FUNCTION_BLOCK Fb_FaultHandler
VAR_INPUT
END_VAR
VAR_OUTPUT
	arActiveFaults 	: ARRAY [0..Param_Messages.nMAX_MESSAGES_SHOWN] OF UDT_Fault  ; // reference to active fault array
	nActiveFaults	: UDINT 			; // reference to active fault counter
	bActOM 			: BOOL := FALSE ;
	bActMC 			: BOOL := FALSE ;
	bActCF 			: BOOL := FALSE ;
	bActFF 			: BOOL := FALSE ;
END_VAR
VAR
	bResetting		: BOOL := FALSE ;
	// functional variables
	i 					: UDINT ;
	// fault data
	stFaultUdt 			: UDT_Fault ;
	bTimedOut 			: BOOL ; // Message has timed out
	// Message logging
	dToday				: DATE ; 
	nWriteStep			: UDINT := 0 ;
	bWriteError			: BOOL 	; // write to file error occured
	nWriteErroId		: UDINT ; // write error id
	// Write variables
	sActFileName		: STRING ;
	hFile				: UINT	:= 0;(* File handle of the source file *)
	sMessageString		: ARRAY [0..Param_Messages.nMESSAGE_COLUMNS] OF STRING (GVL_Parameters.MAX_CSV_FIELD_LENGTH); (* temporary parameter buffer to string*)
	sCSVLine			: T_MaxString := '';(* Single CSV text line (row, record), we are using string as record buffer (your are able to see created fields) *)
	sCSVField			: T_MaxString := '';(* Single CSV field value (column, record field) *)

	// Log to file functions
	fbFileOpen		: FB_FileOpen	;(* Opens file *)
	fbFileClose		: FB_FileClose	;(* Closes file *)
	fbFileGets		: FB_FileGets	;(* Reads one record (line) *)
	fbFilePuts		: FB_FilePuts	;(* Writes one record (line) *)
	fbReader		: FB_CSVMemBufferReader;(* Helper function block used to parse CSV data bytes (single record line) *)
	fbWriter		: FB_CSVMemBufferWriter;(* Helper function block used to create CSV data bytes (single record line) *)
END_VAR
VAR PERSISTENT
	dLastFileDate : DATE ;
END_VAR
VAR CONSTANT
	stEmptyMessageUdt : UDT_Fault := (	Active 			:= FALSE,
										FaultType 		:= E_FaultTypes.NA,
										MessageNumber	:= 0,
										LocationNumber	:= 0,
										Discription 	:= '',
										LocationName	:= '',
										ComponentType	:= E_ComponentTypes.NA,
										StartTime		:= DT#2020-1-1-00:00:00,
										EndTime			:= DT#2020-1-1-00:00:00,
										FullFaultId		:= '0'	)  ;
END_VAR

// Check for active faults in list
IF NOT bResetting THEN 
	ExecSetFaultBit(); 
END_IF

bResetting := FALSE ;

METHOD PRIVATE CheckEntryValid : BOOL
VAR_IN_OUT
	stFault : UDT_Fault ; // actuive fault structure input
END_VAR
VAR
	// functional variables
	i 	: UDINT ;
END_VAR
// ======= check if new entry is valid and not already active ======
CheckEntryValid S= TRUE ;
FOR i := 0 TO nActiveFaults DO
	IF arActiveFaults[i].Discription = stFault.Discription THEN 
		CheckEntryValid 			:= FALSE ; 
		arActiveFaults[i].Active 	:= TRUE ; 
	END_IF
END_FOR
END_METHOD

METHOD PUBLIC CmdAddFault : BOOL
VAR_IN_OUT
	stFault : UDT_Fault ; // active fault structure input
END_VAR
// coppy fault to internal fault udt
IF stFault.FaultType <> E_FaultTypes.NA AND stFault.Active THEN 
	// Process fault data
	IF CheckEntryValid(stFault) AND NOT bResetting THEN
		THIS^.stFaultUdt	:= stFault ;
		ExecWriteMessage();
	END_IF
	stFault 			:= stEmptyMessageUdt ;
	stFaultUdt.Active	:= FALSE ;
END_IF
END_METHOD

METHOD PUBLIC CmdReset : BOOL
VAR_INPUT
END_VAR
bResetting := TRUE ;
// Check for reset is active 
CmdReset := ExecResetFaults();
END_METHOD

METHOD PRIVATE ExecCleanUpArray : BOOL
VAR
	// functional variables
	i 					: UDINT ;
END_VAR
// Clean up array by removing blanc spaces 
FOR i := 0 TO Param_Messages.nMAX_MESSAGES_SHOWN - 1 DO 
	IF arActiveFaults[i].FaultType = 0 THEN 
		arActiveFaults[i] 	:= arActiveFaults[i+1];
		arActiveFaults[i+1] := stEmptyMessageUdt;
	END_IF
END_FOR

//Sort messages after cleaning
ExecSortMessages();
END_METHOD

METHOD PRIVATE ExecResetFaults : BOOL
VAR
	nResetPoint : UDINT := 0 ; // point of reset for active fault array (skips fault if .active bit is true)
	// functional variables
	i 					: UDINT ;
END_VAR
FOR i := 0 TO Param_Messages.nMAX_MESSAGES_SHOWN DO
	IF arActiveFaults[i].Active THEN
		CONTINUE;
	ELSE
		arActiveFaults[i] := stEmptyMessageUdt; 
	END_IF
END_FOR

ExecCleanUpArray();

bActOM 			:= FALSE;
bActMC 			:= FALSE;
bActCF 			:= FALSE;
bActFF 			:= FALSE;

ExecResetFaults := TRUE ;
END_METHOD

METHOD PRIVATE ExecSetFaultBit : BOOL
bActOM 	:= FALSE;
bActMC	:= FALSE;
bActCF 	:= FALSE;
bActFF 	:= FALSE;
	
FOR i := 0 TO nActiveFaults DO
	// read message type 
	CASE arActiveFaults[i].FaultType OF
		E_FaultTypes.OM : 
			IF arActiveFaults[i].Active THEN 
				bActOM 		S= TRUE ;
				
			ELSE 
				bTimedOut 	S= TRUE ;
			END_IF 
		E_FaultTypes.MC :
			IF arActiveFaults[i].Active THEN 
				bActMC 		S= TRUE ;
			ELSE 
				bTimedOut 	S= TRUE ;
			END_IF 
		E_FaultTypes.CF:
			bActCF 		S= TRUE ;
		E_FaultTypes.FF:
			bActFF 		S= TRUE ;
		ELSE
			bTimedOut := FALSE ;
	END_CASE

	IF bTimedOut THEN 
		arActiveFaults[i] := stEmptyMessageUdt;				
		bTimedOut := FALSE ;
	END_IF
	// Reset active bit when timed out, if fault is still active it will be set to true again.
	arActiveFaults[i].Active R= (arActiveFaults[i].StartTime + Param_Messages.tMESSAGE_TIMEOUT) < Sys_Variables.SystemTime;
END_FOR

// clean up the fault array
ExecCleanUpArray();
END_METHOD

METHOD INTERNAL ExecSortMessages : BOOL
VAR
	k : UDINT ;
	stTempMessageStorage : UDT_Fault ; // Temporary message storage for sorting
END_VAR
FOR k := 1 TO Param_Messages.nMAX_MESSAGES_SHOWN - 1 DO 
	FOR i := 0 TO Param_Messages.nMAX_MESSAGES_SHOWN - 2 DO 
		IF arActiveFaults[i].FaultType < arActiveFaults[i+1].FaultType THEN 
			stTempMessageStorage 	:= arActiveFaults[i];
			arActiveFaults[i]		:= arActiveFaults[i+1];
			arActiveFaults[i+1]		:= stTempMessageStorage;
		END_IF
	END_FOR	 
END_FOR

ExecSortMessages := TRUE;
END_METHOD

ACTION ExecWriteMessage:
// Set message start time 
stFaultUdt.StartTime := Sys_Variables.SystemTime ;
// Fill Full Fault Id
stFaultUdt.FullFaultId := TO_STRING(stFaultUdt.FaultType);
stFaultUdt.FullFaultId := CONCAT(stFaultUdt.FullFaultId,'.');
stFaultUdt.FullFaultId := CONCAT(stFaultUdt.FullFaultId,UDINT_TO_STRING(stFaultUdt.MessageNumber));
stFaultUdt.FullFaultId := CONCAT(stFaultUdt.FullFaultId,'.');
stFaultUdt.FullFaultId := CONCAT(stFaultUdt.FullFaultId,UDINT_TO_STRING(stFaultUdt.LocationNumber));
stFaultUdt.FullFaultId := CONCAT(stFaultUdt.FullFaultId,'.');
stFaultUdt.FullFaultId := CONCAT(stFaultUdt.FullFaultId,UDINT_TO_STRING(stFaultUdt.ComponentType));
// send message to higher level 
arActiveFaults[nActiveFaults] := stFaultUdt		;
// Sort shown Massages
ExecSortMessages();
// Set pointer to next fault
IF nActiveFaults < Param_Messages.nMAX_MESSAGES_SHOWN THEN 
	nActiveFaults := nActiveFaults + 1 	;
ELSE
	nActiveFaults := 0 ;
END_IF

// Sort Messages by severity
END_ACTION

END_FUNCTION_BLOCK

(* stored: Version 1.1.0.1, ProductVersion 3.1.4024.10
   POU Fb_FaultHandler: Id {08f65884-c647-4a29-b7ba-51d088979c07}, SpecialFunc None
   Folder Private: Id {2e728eb6-79bc-4de8-8875-9d08a8df9edd}
   Method CheckEntryValid: Id {4ead88ed-0ad4-4581-8230-d979907ffe1b}
   Method CmdAddFault: Id {cd103280-aca4-4b4a-a070-10b84eec5ffb}
   Method CmdReset: Id {a9c5d6bc-61dd-41fc-99d9-5b14d5fa2712}
   Method ExecCleanUpArray: Id {f3ade57a-1ab7-4952-98ed-276828beb548}
   Method ExecResetFaults: Id {69b2b7d1-18ff-442a-8c8e-bfbea5c9f66f}
   Method ExecSetFaultBit: Id {1d4b6758-0786-425a-a6f8-dc8178d0967d}
   Method ExecSortMessages: Id {9379339c-5f6e-4e04-abc6-6a8505afc20b}
   Action ExecWriteMessage: Id {3af8b3ee-c7f9-4b45-bd33-128a18baf300} *)
